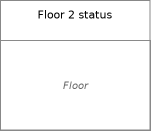
VISUALIZATION Screen2  // 151x131
    Frame (0,40 151x91)
        shows Floor(LS_Floor := MAIN.LS_Floor[2])
        OnMouseClick: change screen: Previous 
    Label (0,0 150x30), "Floor 2 status"
END_VISUALIZATION

(* stored: Version 1.1.0.1, ProductVersion 3.1.4024.11
   Visu Screen2: Id {3c4dae1f-e6f2-4b7c-9e0d-1d7b3391f7d9} *)
